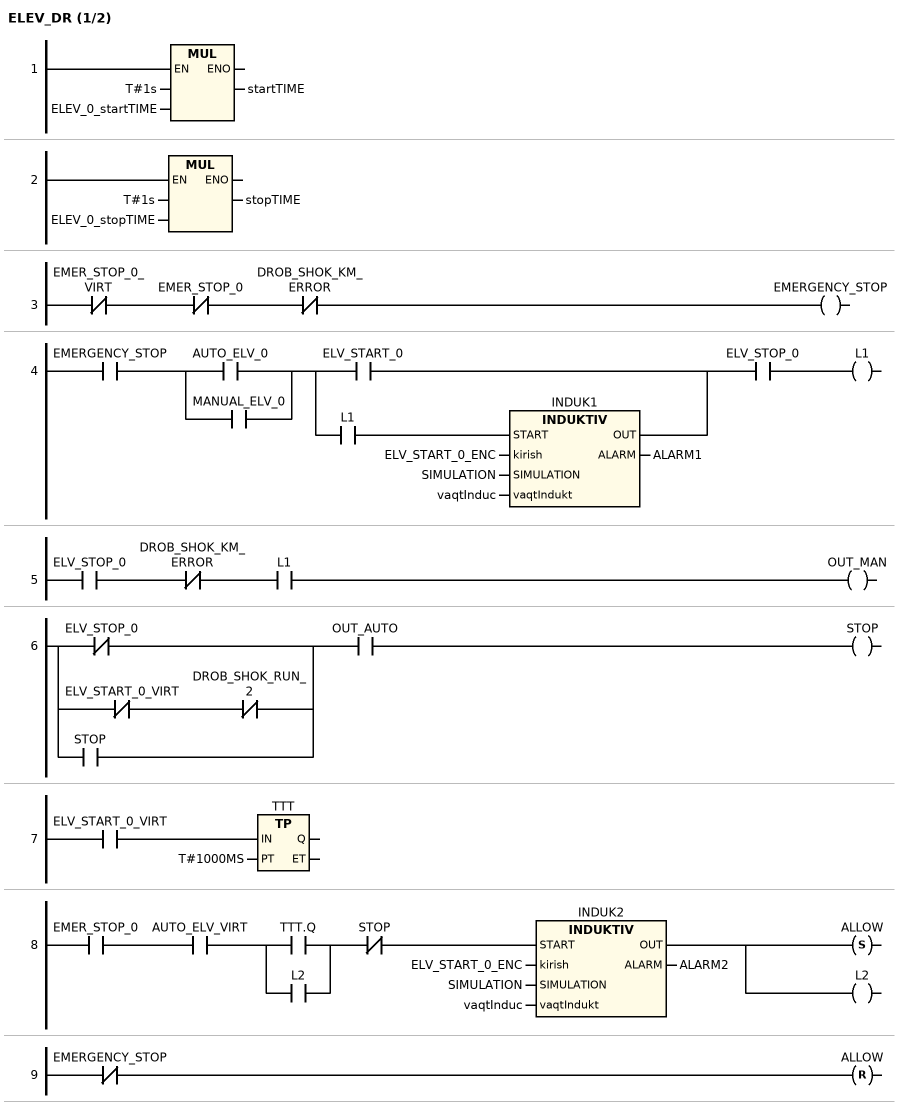
[picture p48: ELEV_DR (LD)]
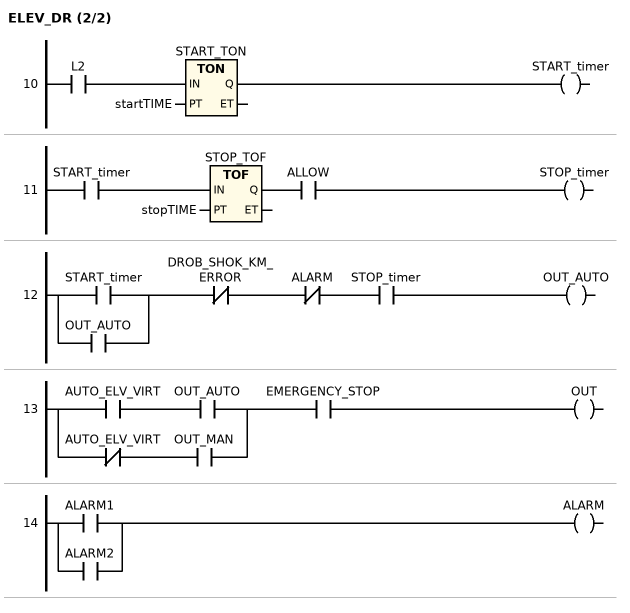
_LD_ (* Ladder Diagram *)
NETWORK 1
	*
		EN --- MUL(T#1s, ELEV_0_startTIME) => startTIME
NETWORK 2
	*
		EN --- MUL(T#1s, ELEV_0_stopTIME) => stopTIME
NETWORK 3
	[/EMER_STOP_0_VIRT] - [/EMER_STOP_0] - [/DROB_SHOK_KM_ERROR] --- (EMERGENCY_STOP)
NETWORK 4
	[EMERGENCY_STOP] - { [AUTO_ELV_0] | [MANUAL_ELV_0] } - { [ELV_START_0] | [L1] - INDUK1:INDUKTIV(START: *, kirish: ELV_START_0_ENC, SIMULATION: SIMULATION, vaqtIndukt: vaqtInduc, ALARM => ALARM1) } - [ELV_STOP_0] --- (L1)
NETWORK 5
	[ELV_STOP_0] - [/DROB_SHOK_KM_ERROR] - [L1] --- (OUT_MAN)
NETWORK 6
	{ [/ELV_STOP_0] | [/ELV_START_0_VIRT] - [/DROB_SHOK_RUN_2] | [STOP] } - [OUT_AUTO] --- (STOP)
NETWORK 7
	[ELV_START_0_VIRT] - TTT:TP(IN: *, PT: T#1000MS)
NETWORK 8
	[EMER_STOP_0] - [AUTO_ELV_VIRT] - { [TTT.Q] | [L2] } - [/STOP] - INDUK2:INDUKTIV(START: *, kirish: ELV_START_0_ENC, SIMULATION: SIMULATION, vaqtIndukt: vaqtInduc, ALARM => ALARM2) --- (S ALLOW) (L2)
NETWORK 9
	[/EMERGENCY_STOP] --- (R ALLOW)
NETWORK 10
	[L2] - START_TON:TON(IN: *, PT: startTIME) --- (START_timer)
NETWORK 11
	[START_timer] - STOP_TOF:TOF(IN: *, PT: stopTIME) - [ALLOW] --- (STOP_timer)
NETWORK 12
	{ [START_timer] | [OUT_AUTO] } - [/DROB_SHOK_KM_ERROR] - [/ALARM] - [STOP_timer] --- (OUT_AUTO)
NETWORK 13
	{ [AUTO_ELV_VIRT] - [OUT_AUTO] | [/AUTO_ELV_VIRT] - [OUT_MAN] } - [EMERGENCY_STOP] --- (OUT)
NETWORK 14
	{ [ALARM1] | [ALARM2] } --- (ALARM)
_END_LD_
(* the same logic as Structured Text *)
(* Network 1 *)
startTIME := T#1s * ELEV_0_startTIME;
(* Network 2 *)
stopTIME := T#1s * ELEV_0_stopTIME;
(* Network 3 *)
EMERGENCY_STOP := NOT EMER_STOP_0_VIRT AND NOT EMER_STOP_0 AND NOT DROB_SHOK_KM_ERROR;
(* Network 4 *)
_p1 := EMERGENCY_STOP AND (AUTO_ELV_0 OR MANUAL_ELV_0);
INDUK1(START := _p1 AND L1, kirish := ELV_START_0_ENC, SIMULATION := SIMULATION, vaqtIndukt := vaqtInduc);
ALARM1 := INDUK1.ALARM;
L1 := (_p1 AND ELV_START_0 OR INDUK1.OUT) AND ELV_STOP_0;
(* Network 5 *)
OUT_MAN := ELV_STOP_0 AND NOT DROB_SHOK_KM_ERROR AND L1;
(* Network 6 *)
STOP := (NOT ELV_STOP_0 OR NOT ELV_START_0_VIRT AND NOT DROB_SHOK_RUN_2 OR STOP) AND OUT_AUTO;
(* Network 7 *)
TTT(IN := ELV_START_0_VIRT, PT := T#1000MS);
(* Network 8 *)
INDUK2(START := EMER_STOP_0 AND AUTO_ELV_VIRT AND (TTT.Q OR L2) AND NOT STOP, kirish := ELV_START_0_ENC, SIMULATION := SIMULATION, vaqtIndukt := vaqtInduc);
ALARM2 := INDUK2.ALARM;
IF INDUK2.OUT THEN ALLOW := TRUE; END_IF;
L2 := INDUK2.OUT;
(* Network 9 *)
IF NOT EMERGENCY_STOP THEN ALLOW := FALSE; END_IF;
(* Network 10 *)
START_TON(IN := L2, PT := startTIME);
START_timer := START_TON.Q;
(* Network 11 *)
STOP_TOF(IN := START_timer, PT := stopTIME);
STOP_timer := STOP_TOF.Q AND ALLOW;
(* Network 12 *)
OUT_AUTO := (START_timer OR OUT_AUTO) AND NOT DROB_SHOK_KM_ERROR AND NOT ALARM AND STOP_timer;
(* Network 13 *)
OUT := (AUTO_ELV_VIRT AND OUT_AUTO OR NOT AUTO_ELV_VIRT AND OUT_MAN) AND EMERGENCY_STOP;
(* Network 14 *)
ALARM := ALARM1 OR ALARM2;
END_FUNCTION_BLOCK

(* POU DROBILKA2, LD *)
PROGRAM DROBILKA2
VAR
	convTON : TON;
	conVAQT : TIME := T#180s;
	drobTON : TON;
	drobVAQT: TIME := T#180s;
	maxTON : TON;
	maxVAQT: TIME := T#5s;
	ELV_F_TRIG: F_TRIG;
	TANK_FULL: BOOL;
	ELV_R_TRIG: R_TRIG;
END_VAR
VAR (* helpers for the ST form of the networks *)
	_p1 : BOOL;
END_VAR
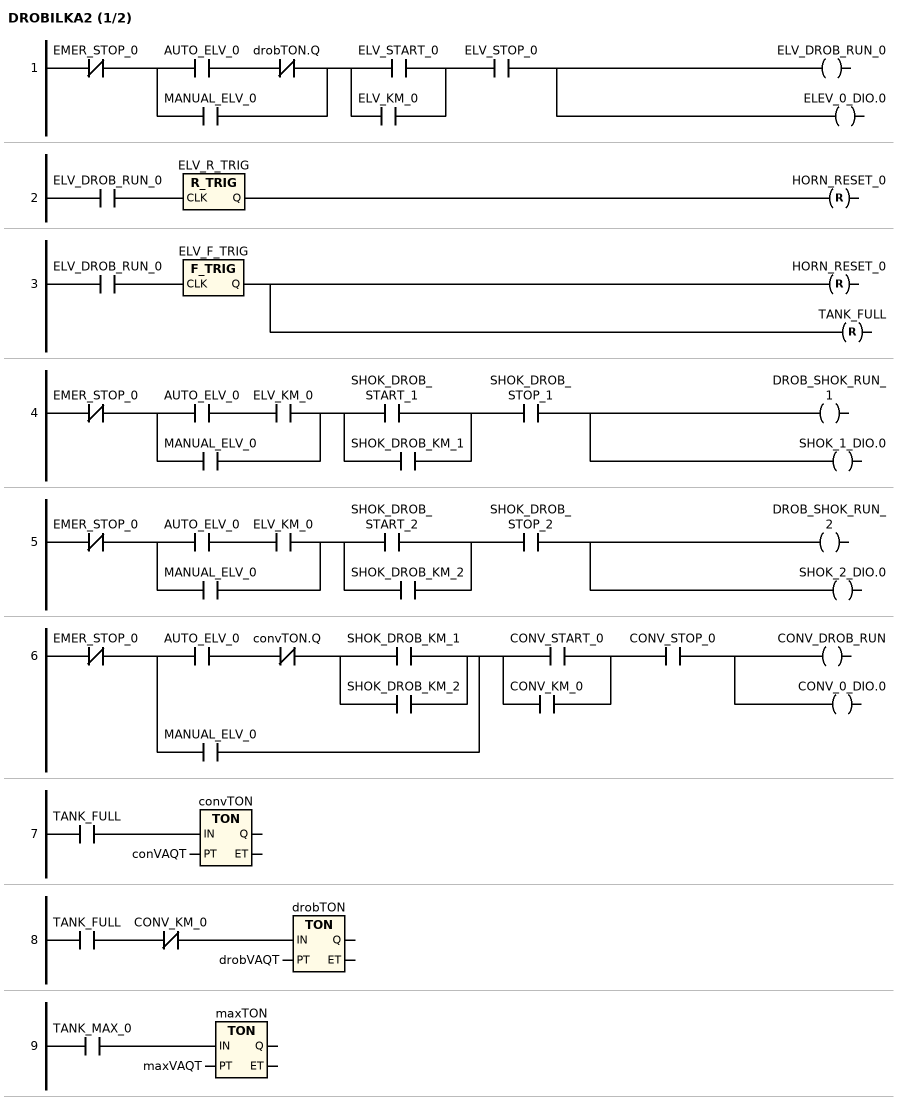
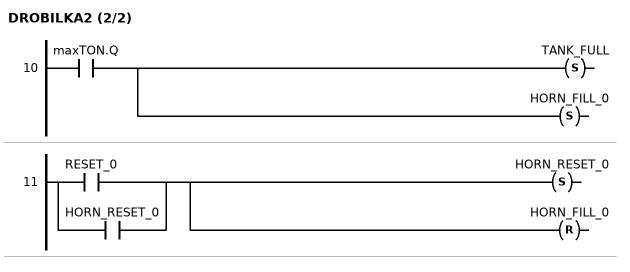
_LD_ (* Ladder Diagram *)
NETWORK 1
	[/EMER_STOP_0] - { [AUTO_ELV_0] - [/drobTON.Q] | [MANUAL_ELV_0] } - { [ELV_START_0] | [ELV_KM_0] } - [ELV_STOP_0] --- (ELV_DROB_RUN_0) (ELEV_0_DIO.0)
NETWORK 2
	[ELV_DROB_RUN_0] - ELV_R_TRIG:R_TRIG(CLK: *) --- (R HORN_RESET_0)
NETWORK 3
	[ELV_DROB_RUN_0] - ELV_F_TRIG:F_TRIG(CLK: *) --- (R HORN_RESET_0) (R TANK_FULL)
NETWORK 4
	[/EMER_STOP_0] - { [AUTO_ELV_0] - [ELV_KM_0] | [MANUAL_ELV_0] } - { [SHOK_DROB_START_1] | [SHOK_DROB_KM_1] } - [SHOK_DROB_STOP_1] --- (DROB_SHOK_RUN_1) (SHOK_1_DIO.0)
NETWORK 5
	[/EMER_STOP_0] - { [AUTO_ELV_0] - [ELV_KM_0] | [MANUAL_ELV_0] } - { [SHOK_DROB_START_2] | [SHOK_DROB_KM_2] } - [SHOK_DROB_STOP_2] --- (DROB_SHOK_RUN_2) (SHOK_2_DIO.0)
NETWORK 6
	[/EMER_STOP_0] - { [AUTO_ELV_0] - [/convTON.Q] - { [SHOK_DROB_KM_1] | [SHOK_DROB_KM_2] } | [MANUAL_ELV_0] } - { [CONV_START_0] | [CONV_KM_0] } - [CONV_STOP_0] --- (CONV_DROB_RUN) (CONV_0_DIO.0)
NETWORK 7
	[TANK_FULL] - convTON:TON(IN: *, PT: conVAQT)
NETWORK 8
	[TANK_FULL] - [/CONV_KM_0] - drobTON:TON(IN: *, PT: drobVAQT)
NETWORK 9
	[TANK_MAX_0] - maxTON:TON(IN: *, PT: maxVAQT)
NETWORK 10
	[maxTON.Q] --- (S TANK_FULL) (S HORN_FILL_0)
NETWORK 11
	{ [RESET_0] | [HORN_RESET_0] } --- (S HORN_RESET_0) (R HORN_FILL_0)
_END_LD_
(* the same logic as Structured Text *)
(* Network 1 *)
ELV_DROB_RUN_0 := NOT EMER_STOP_0 AND (AUTO_ELV_0 AND NOT drobTON.Q OR MANUAL_ELV_0) AND (ELV_START_0 OR ELV_KM_0) AND ELV_STOP_0;
ELEV_0_DIO.0 := ELV_DROB_RUN_0;
(* Network 2 *)
ELV_R_TRIG(CLK := ELV_DROB_RUN_0);
IF ELV_R_TRIG.Q THEN HORN_RESET_0 := FALSE; END_IF;
(* Network 3 *)
ELV_F_TRIG(CLK := ELV_DROB_RUN_0);
IF ELV_F_TRIG.Q THEN HORN_RESET_0 := FALSE; TANK_FULL := FALSE; END_IF;
(* Network 4 *)
DROB_SHOK_RUN_1 := NOT EMER_STOP_0 AND (AUTO_ELV_0 AND ELV_KM_0 OR MANUAL_ELV_0) AND (SHOK_DROB_START_1 OR SHOK_DROB_KM_1) AND SHOK_DROB_STOP_1;
SHOK_1_DIO.0 := DROB_SHOK_RUN_1;
(* Network 5 *)
DROB_SHOK_RUN_2 := NOT EMER_STOP_0 AND (AUTO_ELV_0 AND ELV_KM_0 OR MANUAL_ELV_0) AND (SHOK_DROB_START_2 OR SHOK_DROB_KM_2) AND SHOK_DROB_STOP_2;
SHOK_2_DIO.0 := DROB_SHOK_RUN_2;
(* Network 6 *)
CONV_DROB_RUN := NOT EMER_STOP_0 AND (AUTO_ELV_0 AND NOT convTON.Q AND (SHOK_DROB_KM_1 OR SHOK_DROB_KM_2) OR MANUAL_ELV_0) AND (CONV_START_0 OR CONV_KM_0) AND CONV_STOP_0;
CONV_0_DIO.0 := CONV_DROB_RUN;
(* Network 7 *)
convTON(IN := TANK_FULL, PT := conVAQT);
(* Network 8 *)
drobTON(IN := TANK_FULL AND NOT CONV_KM_0, PT := drobVAQT);
(* Network 9 *)
maxTON(IN := TANK_MAX_0, PT := maxVAQT);
(* Network 10 *)
IF maxTON.Q THEN TANK_FULL := TRUE; HORN_FILL_0 := TRUE; END_IF;
(* Network 11 *)
_p1 := RESET_0 OR HORN_RESET_0;
IF _p1 THEN HORN_RESET_0 := TRUE; HORN_FILL_0 := FALSE; END_IF;
END_PROGRAM

(* POU main_1212, LD *)
PROGRAM main_1212
VAR
	MAH_YET3 : BOOL;
	VAQT : TIME := T#10s;
       VAQT1: TIME := T#4s;
       VAQT2 : TIME := T#6s;
      VAQT3 : TIME := T#6s;
	vaqtInduc : WORD := 15;
	VIBRATOR3_T: BOOL;
	TON1: TON;
	TON2: TON;
	OUT: BOOL;
	IND1: INDUKTIV;
	IND2: INDUKTIV;


	STOP: BOOL;
	CHIQSH: BOOL;
	PUSK: BOOL;
	MAH_YET4: BOOL;
	VIBRATOR4_T: BOOL;
	induk: BOOL;

	ALR_ELEV1: BOOL;
	ALR_ELEV2: BOOL;
	ALR_ELEV3: BOOL;
	ALR_ELEV4: BOOL;
	IND_ELV_1: INDUKTIV;
	IND_SHNK_3: INDUKTIV;
	IND_SHNK_4: INDUKTIV;
	IND_SHNK_SKL_4: INDUKTIV;
	IND_SEPR_4: INDUKTIV;
	IND_MILL_3: INDUKTIV;
	IND_MILL_4: INDUKTIV;

END_VAR
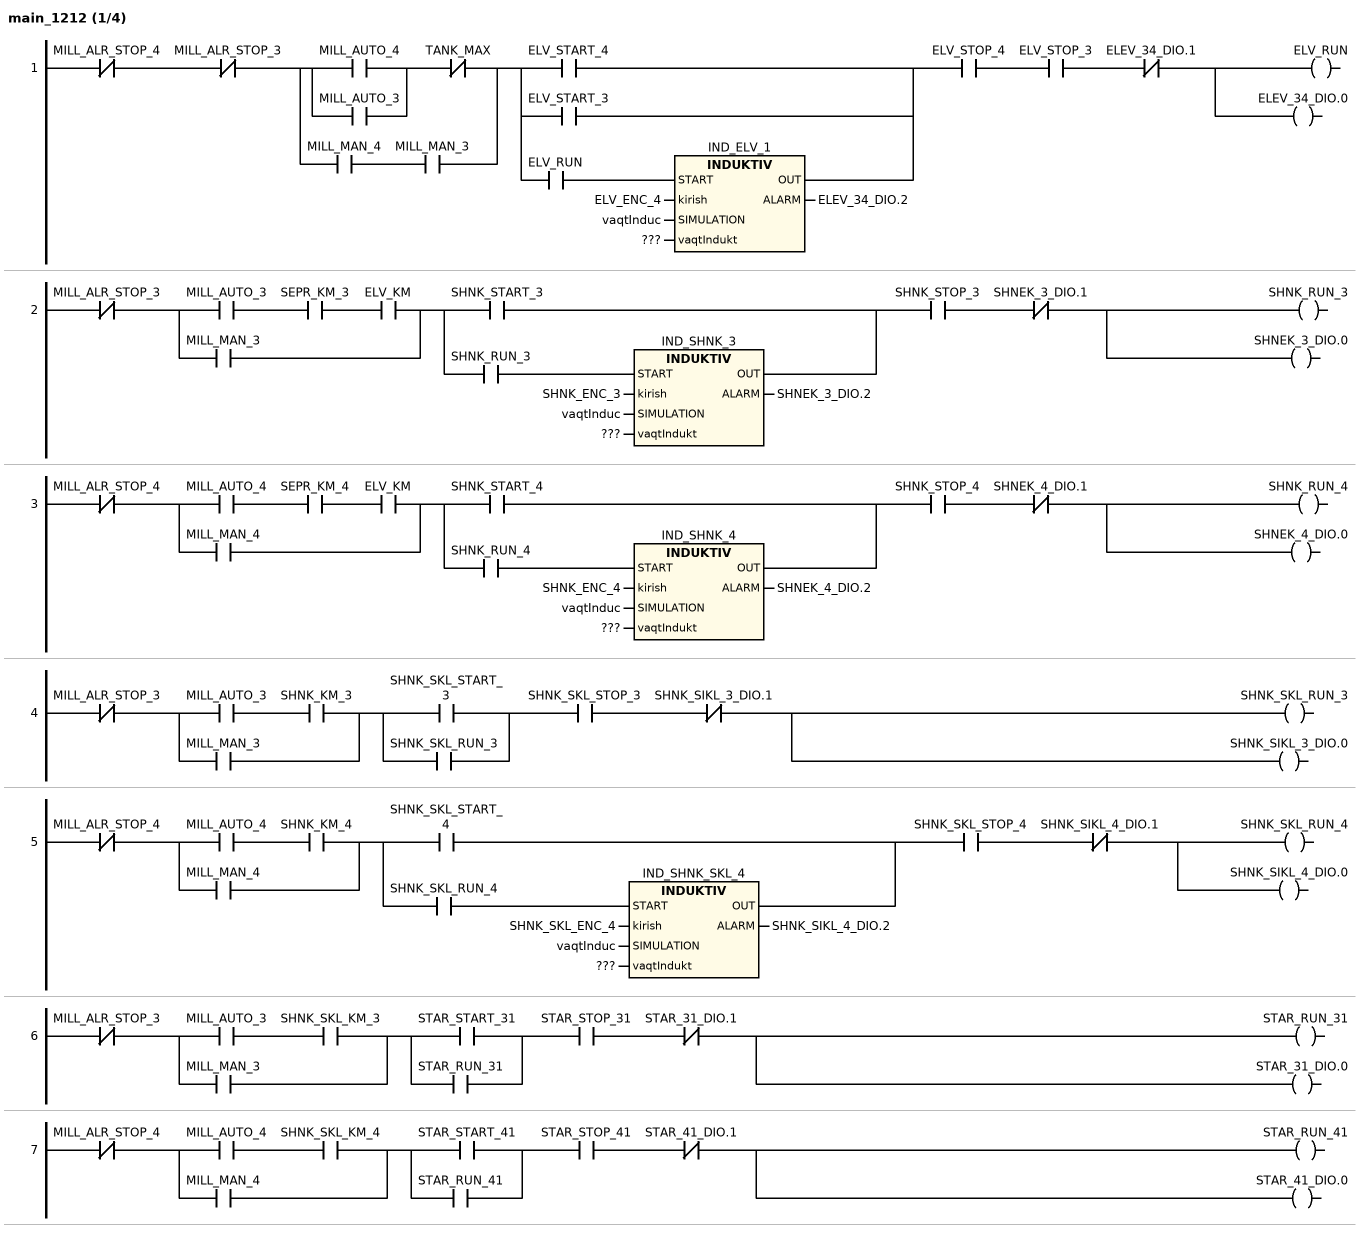
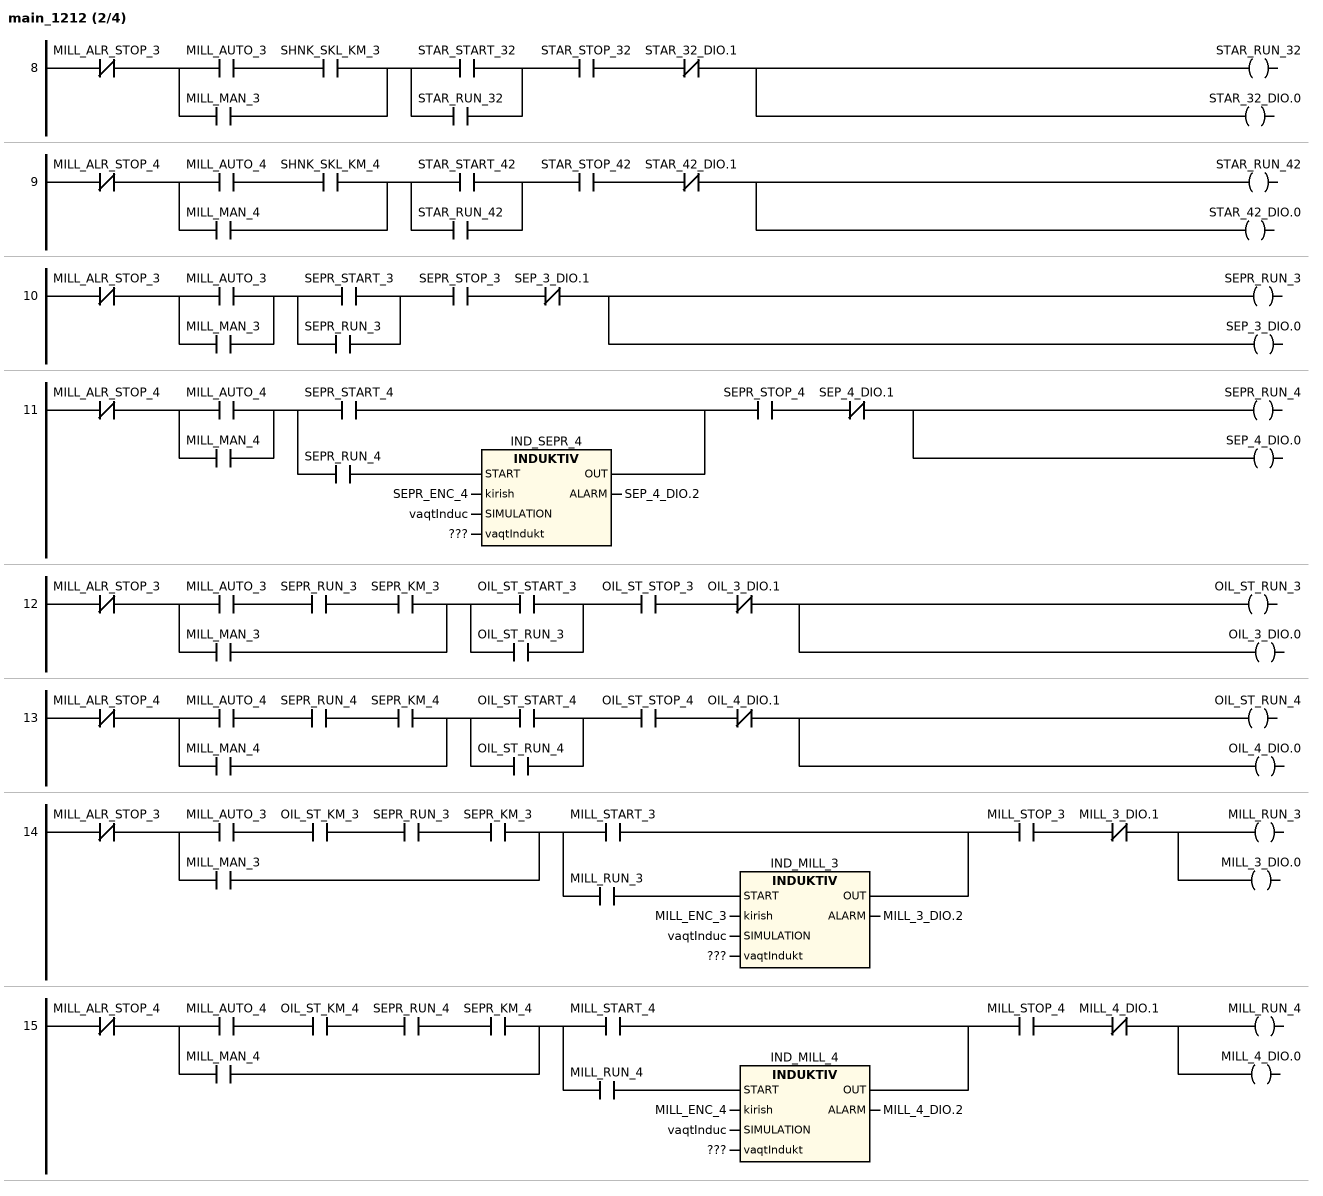
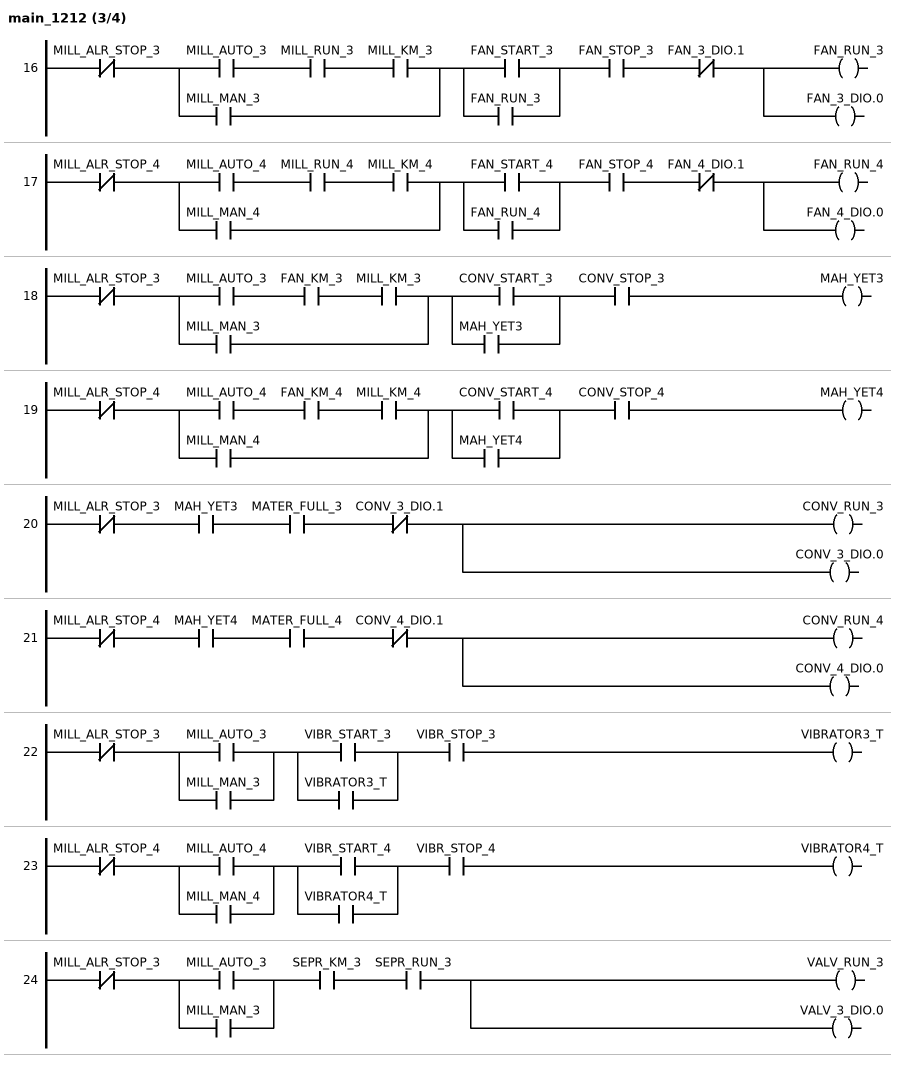
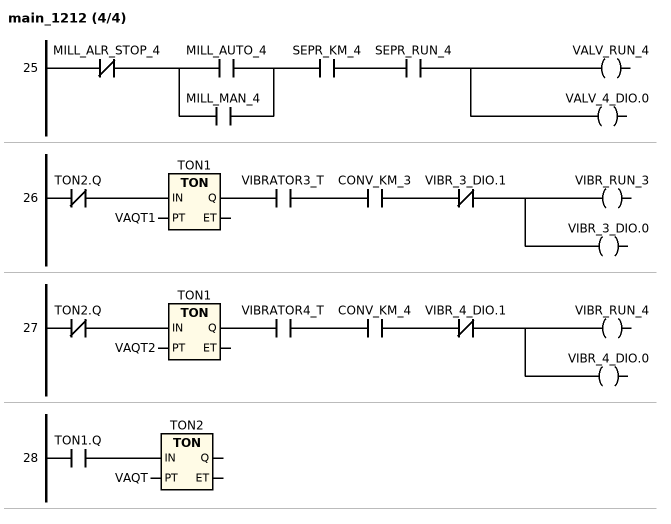
_LD_ (* Ladder Diagram *)
NETWORK 1
	[/MILL_ALR_STOP_4] - [/MILL_ALR_STOP_3] - { { [MILL_AUTO_4] | [MILL_AUTO_3] } - [/TANK_MAX] | [MILL_MAN_4] - [MILL_MAN_3] } - { [ELV_START_4] | [ELV_START_3] | [ELV_RUN] - IND_ELV_1:INDUKTIV(START: *, kirish: ELV_ENC_4, SIMULATION: vaqtInduc, vaqtIndukt: ???, ALARM => ELEV_34_DIO.2) } - [ELV_STOP_4] - [ELV_STOP_3] - [/ELEV_34_DIO.1] --- (ELV_RUN) (ELEV_34_DIO.0)
NETWORK 2
	[/MILL_ALR_STOP_3] - { [MILL_AUTO_3] - [SEPR_KM_3] - [ELV_KM] | [MILL_MAN_3] } - { [SHNK_START_3] | [SHNK_RUN_3] - IND_SHNK_3:INDUKTIV(START: *, kirish: SHNK_ENC_3, SIMULATION: vaqtInduc, vaqtIndukt: ???, ALARM => SHNEK_3_DIO.2) } - [SHNK_STOP_3] - [/SHNEK_3_DIO.1] --- (SHNK_RUN_3) (SHNEK_3_DIO.0)
NETWORK 3
	[/MILL_ALR_STOP_4] - { [MILL_AUTO_4] - [SEPR_KM_4] - [ELV_KM] | [MILL_MAN_4] } - { [SHNK_START_4] | [SHNK_RUN_4] - IND_SHNK_4:INDUKTIV(START: *, kirish: SHNK_ENC_4, SIMULATION: vaqtInduc, vaqtIndukt: ???, ALARM => SHNEK_4_DIO.2) } - [SHNK_STOP_4] - [/SHNEK_4_DIO.1] --- (SHNK_RUN_4) (SHNEK_4_DIO.0)
NETWORK 4
	[/MILL_ALR_STOP_3] - { [MILL_AUTO_3] - [SHNK_KM_3] | [MILL_MAN_3] } - { [SHNK_SKL_START_3] | [SHNK_SKL_RUN_3] } - [SHNK_SKL_STOP_3] - [/SHNK_SIKL_3_DIO.1] --- (SHNK_SKL_RUN_3) (SHNK_SIKL_3_DIO.0)
NETWORK 5
	[/MILL_ALR_STOP_4] - { [MILL_AUTO_4] - [SHNK_KM_4] | [MILL_MAN_4] } - { [SHNK_SKL_START_4] | [SHNK_SKL_RUN_4] - IND_SHNK_SKL_4:INDUKTIV(START: *, kirish: SHNK_SKL_ENC_4, SIMULATION: vaqtInduc, vaqtIndukt: ???, ALARM => SHNK_SIKL_4_DIO.2) } - [SHNK_SKL_STOP_4] - [/SHNK_SIKL_4_DIO.1] --- (SHNK_SKL_RUN_4) (SHNK_SIKL_4_DIO.0)
NETWORK 6
	[/MILL_ALR_STOP_3] - { [MILL_AUTO_3] - [SHNK_SKL_KM_3] | [MILL_MAN_3] } - { [STAR_START_31] | [STAR_RUN_31] } - [STAR_STOP_31] - [/STAR_31_DIO.1] --- (STAR_RUN_31) (STAR_31_DIO.0)
NETWORK 7
	[/MILL_ALR_STOP_4] - { [MILL_AUTO_4] - [SHNK_SKL_KM_4] | [MILL_MAN_4] } - { [STAR_START_41] | [STAR_RUN_41] } - [STAR_STOP_41] - [/STAR_41_DIO.1] --- (STAR_RUN_41) (STAR_41_DIO.0)
NETWORK 8
	[/MILL_ALR_STOP_3] - { [MILL_AUTO_3] - [SHNK_SKL_KM_3] | [MILL_MAN_3] } - { [STAR_START_32] | [STAR_RUN_32] } - [STAR_STOP_32] - [/STAR_32_DIO.1] --- (STAR_RUN_32) (STAR_32_DIO.0)
NETWORK 9
	[/MILL_ALR_STOP_4] - { [MILL_AUTO_4] - [SHNK_SKL_KM_4] | [MILL_MAN_4] } - { [STAR_START_42] | [STAR_RUN_42] } - [STAR_STOP_42] - [/STAR_42_DIO.1] --- (STAR_RUN_42) (STAR_42_DIO.0)
NETWORK 10
	[/MILL_ALR_STOP_3] - { [MILL_AUTO_3] | [MILL_MAN_3] } - { [SEPR_START_3] | [SEPR_RUN_3] } - [SEPR_STOP_3] - [/SEP_3_DIO.1] --- (SEPR_RUN_3) (SEP_3_DIO.0)
NETWORK 11
	[/MILL_ALR_STOP_4] - { [MILL_AUTO_4] | [MILL_MAN_4] } - { [SEPR_START_4] | [SEPR_RUN_4] - IND_SEPR_4:INDUKTIV(START: *, kirish: SEPR_ENC_4, SIMULATION: vaqtInduc, vaqtIndukt: ???, ALARM => SEP_4_DIO.2) } - [SEPR_STOP_4] - [/SEP_4_DIO.1] --- (SEPR_RUN_4) (SEP_4_DIO.0)
NETWORK 12
	[/MILL_ALR_STOP_3] - { [MILL_AUTO_3] - [SEPR_RUN_3] - [SEPR_KM_3] | [MILL_MAN_3] } - { [OIL_ST_START_3] | [OIL_ST_RUN_3] } - [OIL_ST_STOP_3] - [/OIL_3_DIO.1] --- (OIL_ST_RUN_3) (OIL_3_DIO.0)
NETWORK 13
	[/MILL_ALR_STOP_4] - { [MILL_AUTO_4] - [SEPR_RUN_4] - [SEPR_KM_4] | [MILL_MAN_4] } - { [OIL_ST_START_4] | [OIL_ST_RUN_4] } - [OIL_ST_STOP_4] - [/OIL_4_DIO.1] --- (OIL_ST_RUN_4) (OIL_4_DIO.0)
NETWORK 14
	[/MILL_ALR_STOP_3] - { [MILL_AUTO_3] - [OIL_ST_KM_3] - [SEPR_RUN_3] - [SEPR_KM_3] | [MILL_MAN_3] } - { [MILL_START_3] | [MILL_RUN_3] - IND_MILL_3:INDUKTIV(START: *, kirish: MILL_ENC_3, SIMULATION: vaqtInduc, vaqtIndukt: ???, ALARM => MILL_3_DIO.2) } - [MILL_STOP_3] - [/MILL_3_DIO.1] --- (MILL_RUN_3) (MILL_3_DIO.0)
NETWORK 15
	[/MILL_ALR_STOP_4] - { [MILL_AUTO_4] - [OIL_ST_KM_4] - [SEPR_RUN_4] - [SEPR_KM_4] | [MILL_MAN_4] } - { [MILL_START_4] | [MILL_RUN_4] - IND_MILL_4:INDUKTIV(START: *, kirish: MILL_ENC_4, SIMULATION: vaqtInduc, vaqtIndukt: ???, ALARM => MILL_4_DIO.2) } - [MILL_STOP_4] - [/MILL_4_DIO.1] --- (MILL_RUN_4) (MILL_4_DIO.0)
NETWORK 16
	[/MILL_ALR_STOP_3] - { [MILL_AUTO_3] - [MILL_RUN_3] - [MILL_KM_3] | [MILL_MAN_3] } - { [FAN_START_3] | [FAN_RUN_3] } - [FAN_STOP_3] - [/FAN_3_DIO.1] --- (FAN_RUN_3) (FAN_3_DIO.0)
NETWORK 17
	[/MILL_ALR_STOP_4] - { [MILL_AUTO_4] - [MILL_RUN_4] - [MILL_KM_4] | [MILL_MAN_4] } - { [FAN_START_4] | [FAN_RUN_4] } - [FAN_STOP_4] - [/FAN_4_DIO.1] --- (FAN_RUN_4) (FAN_4_DIO.0)
NETWORK 18
	[/MILL_ALR_STOP_3] - { [MILL_AUTO_3] - [FAN_KM_3] - [MILL_KM_3] | [MILL_MAN_3] } - { [CONV_START_3] | [MAH_YET3] } - [CONV_STOP_3] --- (MAH_YET3)
NETWORK 19
	[/MILL_ALR_STOP_4] - { [MILL_AUTO_4] - [FAN_KM_4] - [MILL_KM_4] | [MILL_MAN_4] } - { [CONV_START_4] | [MAH_YET4] } - [CONV_STOP_4] --- (MAH_YET4)
NETWORK 20
	[/MILL_ALR_STOP_3] - [MAH_YET3] - [MATER_FULL_3] - [/CONV_3_DIO.1] --- (CONV_RUN_3) (CONV_3_DIO.0)
NETWORK 21
	[/MILL_ALR_STOP_4] - [MAH_YET4] - [MATER_FULL_4] - [/CONV_4_DIO.1] --- (CONV_RUN_4) (CONV_4_DIO.0)
NETWORK 22
	[/MILL_ALR_STOP_3] - { [MILL_AUTO_3] | [MILL_MAN_3] } - { [VIBR_START_3] | [VIBRATOR3_T] } - [VIBR_STOP_3] --- (VIBRATOR3_T)
NETWORK 23
	[/MILL_ALR_STOP_4] - { [MILL_AUTO_4] | [MILL_MAN_4] } - { [VIBR_START_4] | [VIBRATOR4_T] } - [VIBR_STOP_4] --- (VIBRATOR4_T)
NETWORK 24
	[/MILL_ALR_STOP_3] - { [MILL_AUTO_3] | [MILL_MAN_3] } - [SEPR_KM_3] - [SEPR_RUN_3] --- (VALV_RUN_3) (VALV_3_DIO.0)
NETWORK 25
	[/MILL_ALR_STOP_4] - { [MILL_AUTO_4] | [MILL_MAN_4] } - [SEPR_KM_4] - [SEPR_RUN_4] --- (VALV_RUN_4) (VALV_4_DIO.0)
NETWORK 26
	[/TON2.Q] - TON1:TON(IN: *, PT: VAQT1) - [VIBRATOR3_T] - [CONV_KM_3] - [/VIBR_3_DIO.1] --- (VIBR_RUN_3) (VIBR_3_DIO.0)
NETWORK 27
	[/TON2.Q] - TON1:TON(IN: *, PT: VAQT2) - [VIBRATOR4_T] - [CONV_KM_4] - [/VIBR_4_DIO.1] --- (VIBR_RUN_4) (VIBR_4_DIO.0)
NETWORK 28
	[TON1.Q] - TON2:TON(IN: *, PT: VAQT)
_END_LD_
(* the same logic as Structured Text *)
(* Network 1: see the listing above *)
(* Network 2: see the listing above *)
(* Network 3: see the listing above *)
(* Network 4 *)
SHNK_SKL_RUN_3 := NOT MILL_ALR_STOP_3 AND (MILL_AUTO_3 AND SHNK_KM_3 OR MILL_MAN_3) AND (SHNK_SKL_START_3 OR SHNK_SKL_RUN_3) AND SHNK_SKL_STOP_3 AND NOT SHNK_SIKL_3_DIO.1;
SHNK_SIKL_3_DIO.0 := SHNK_SKL_RUN_3;
(* Network 5: see the listing above *)
(* Network 6 *)
STAR_RUN_31 := NOT MILL_ALR_STOP_3 AND (MILL_AUTO_3 AND SHNK_SKL_KM_3 OR MILL_MAN_3) AND (STAR_START_31 OR STAR_RUN_31) AND STAR_STOP_31 AND NOT STAR_31_DIO.1;
STAR_31_DIO.0 := STAR_RUN_31;
(* Network 7 *)
STAR_RUN_41 := NOT MILL_ALR_STOP_4 AND (MILL_AUTO_4 AND SHNK_SKL_KM_4 OR MILL_MAN_4) AND (STAR_START_41 OR STAR_RUN_41) AND STAR_STOP_41 AND NOT STAR_41_DIO.1;
STAR_41_DIO.0 := STAR_RUN_41;
(* Network 8 *)
STAR_RUN_32 := NOT MILL_ALR_STOP_3 AND (MILL_AUTO_3 AND SHNK_SKL_KM_3 OR MILL_MAN_3) AND (STAR_START_32 OR STAR_RUN_32) AND STAR_STOP_32 AND NOT STAR_32_DIO.1;
STAR_32_DIO.0 := STAR_RUN_32;
(* Network 9 *)
STAR_RUN_42 := NOT MILL_ALR_STOP_4 AND (MILL_AUTO_4 AND SHNK_SKL_KM_4 OR MILL_MAN_4) AND (STAR_START_42 OR STAR_RUN_42) AND STAR_STOP_42 AND NOT STAR_42_DIO.1;
STAR_42_DIO.0 := STAR_RUN_42;
(* Network 10 *)
SEPR_RUN_3 := NOT MILL_ALR_STOP_3 AND (MILL_AUTO_3 OR MILL_MAN_3) AND (SEPR_START_3 OR SEPR_RUN_3) AND SEPR_STOP_3 AND NOT SEP_3_DIO.1;
SEP_3_DIO.0 := SEPR_RUN_3;
(* Network 11: see the listing above *)
(* Network 12 *)
OIL_ST_RUN_3 := NOT MILL_ALR_STOP_3 AND (MILL_AUTO_3 AND SEPR_RUN_3 AND SEPR_KM_3 OR MILL_MAN_3) AND (OIL_ST_START_3 OR OIL_ST_RUN_3) AND OIL_ST_STOP_3 AND NOT OIL_3_DIO.1;
OIL_3_DIO.0 := OIL_ST_RUN_3;
(* Network 13 *)
OIL_ST_RUN_4 := NOT MILL_ALR_STOP_4 AND (MILL_AUTO_4 AND SEPR_RUN_4 AND SEPR_KM_4 OR MILL_MAN_4) AND (OIL_ST_START_4 OR OIL_ST_RUN_4) AND OIL_ST_STOP_4 AND NOT OIL_4_DIO.1;
OIL_4_DIO.0 := OIL_ST_RUN_4;
(* Network 14: see the listing above *)
(* Network 15: see the listing above *)
(* Network 16 *)
FAN_RUN_3 := NOT MILL_ALR_STOP_3 AND (MILL_AUTO_3 AND MILL_RUN_3 AND MILL_KM_3 OR MILL_MAN_3) AND (FAN_START_3 OR FAN_RUN_3) AND FAN_STOP_3 AND NOT FAN_3_DIO.1;
FAN_3_DIO.0 := FAN_RUN_3;
(* Network 17 *)
FAN_RUN_4 := NOT MILL_ALR_STOP_4 AND (MILL_AUTO_4 AND MILL_RUN_4 AND MILL_KM_4 OR MILL_MAN_4) AND (FAN_START_4 OR FAN_RUN_4) AND FAN_STOP_4 AND NOT FAN_4_DIO.1;
FAN_4_DIO.0 := FAN_RUN_4;
(* Network 18 *)
MAH_YET3 := NOT MILL_ALR_STOP_3 AND (MILL_AUTO_3 AND FAN_KM_3 AND MILL_KM_3 OR MILL_MAN_3) AND (CONV_START_3 OR MAH_YET3) AND CONV_STOP_3;
(* Network 19 *)
MAH_YET4 := NOT MILL_ALR_STOP_4 AND (MILL_AUTO_4 AND FAN_KM_4 AND MILL_KM_4 OR MILL_MAN_4) AND (CONV_START_4 OR MAH_YET4) AND CONV_STOP_4;
(* Network 20 *)
CONV_RUN_3 := NOT MILL_ALR_STOP_3 AND MAH_YET3 AND MATER_FULL_3 AND NOT CONV_3_DIO.1;
CONV_3_DIO.0 := CONV_RUN_3;
(* Network 21 *)
CONV_RUN_4 := NOT MILL_ALR_STOP_4 AND MAH_YET4 AND MATER_FULL_4 AND NOT CONV_4_DIO.1;
CONV_4_DIO.0 := CONV_RUN_4;
(* Network 22 *)
VIBRATOR3_T := NOT MILL_ALR_STOP_3 AND (MILL_AUTO_3 OR MILL_MAN_3) AND (VIBR_START_3 OR VIBRATOR3_T) AND VIBR_STOP_3;
(* Network 23 *)
VIBRATOR4_T := NOT MILL_ALR_STOP_4 AND (MILL_AUTO_4 OR MILL_MAN_4) AND (VIBR_START_4 OR VIBRATOR4_T) AND VIBR_STOP_4;
(* Network 24 *)
VALV_RUN_3 := NOT MILL_ALR_STOP_3 AND (MILL_AUTO_3 OR MILL_MAN_3) AND SEPR_KM_3 AND SEPR_RUN_3;
VALV_3_DIO.0 := VALV_RUN_3;
(* Network 25 *)
VALV_RUN_4 := NOT MILL_ALR_STOP_4 AND (MILL_AUTO_4 OR MILL_MAN_4) AND SEPR_KM_4 AND SEPR_RUN_4;
VALV_4_DIO.0 := VALV_RUN_4;
(* Network 26 *)
TON1(IN := NOT TON2.Q, PT := VAQT1);
VIBR_RUN_3 := TON1.Q AND VIBRATOR3_T AND CONV_KM_3 AND NOT VIBR_3_DIO.1;
VIBR_3_DIO.0 := VIBR_RUN_3;
(* Network 27 *)
TON1(IN := NOT TON2.Q, PT := VAQT2);
VIBR_RUN_4 := TON1.Q AND VIBRATOR4_T AND CONV_KM_4 AND NOT VIBR_4_DIO.1;
VIBR_4_DIO.0 := VIBR_RUN_4;
(* Network 28 *)
TON2(IN := TON1.Q, PT := VAQT);
END_PROGRAM

(* POU INDUKTIV_2, CFC *)
FUNCTION_BLOCK INDUKTIV_2
VAR_IN_OUT

	(*RESET : BOOL;*)

END_VAR
VAR_INPUT
	START : BOOL;
	kirish : BOOL;
	vaqtIndukt : WORD := 15;
END_VAR

VAR_OUTPUT

	OUT : BOOL;
	ALARM : BOOL;
END_VAR
VAR
	ton1: TON;
	vaqt : TIME;
	ton2: TON;
	TP1: TP;
	TP2: TP;


END_VAR
VAR (* helpers for the ST form of the networks *)
	_t11 : BOOL;
	_t41 : BOOL;
	_t47 : BOOL;
	_t44 : BOOL;
	_t45 : BOOL;
	_en19 : BOOL;
END_VAR
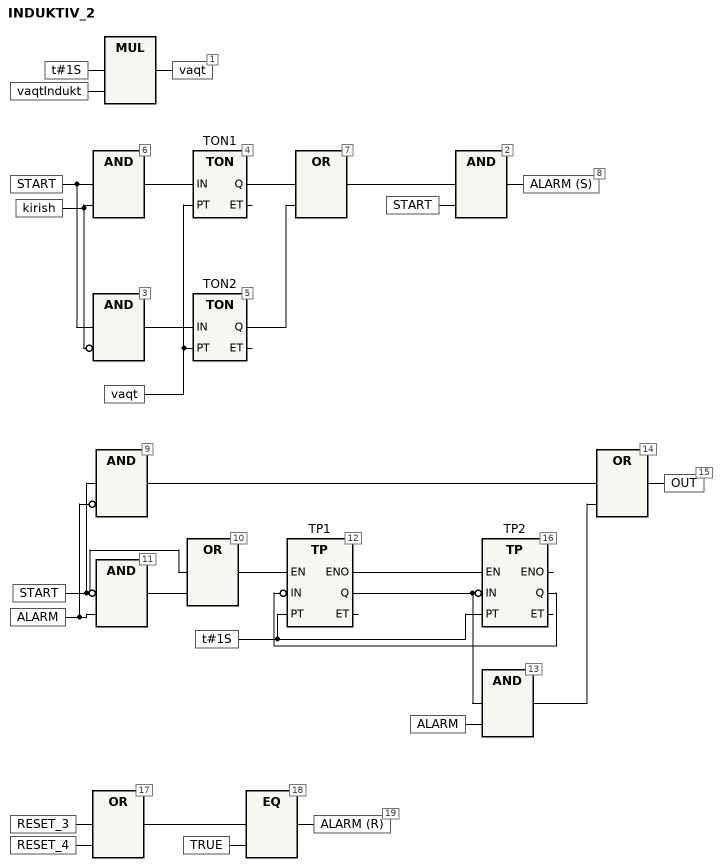
_CFC_ (* Continuous Function Chart, elements in execution order *)
#0 MUL(t#1S, vaqtIndukt)
#1 vaqt <= #0
#2 AND(#7, START)
#3 AND(START, NOT kirish)
#4 TON1:TON(IN: #6, PT: vaqt)
#5 TON2:TON(IN: #3, PT: vaqt)
#6 AND(START, kirish)
#7 OR(#4.Q, #5.Q)
#8 S ALARM <= #2
#9 AND(START, NOT ALARM)
#10 OR(START, #11)
#11 AND(NOT START, ALARM)
#12 TP1:TP(EN: #10, IN: NOT #16.Q, PT: t#1S)
#13 AND(#12.Q, ALARM)
#14 OR(#9, #13)
#15 OUT <= #14
#16 TP2:TP(EN: #12.ENO, IN: NOT #12.Q, PT: t#1S)
#17 OR(RESET_3, RESET_4)
#18 EQ(#17, TRUE)
#19 R ALARM <= #18
_END_CFC_
(* the same logic as Structured Text *)
vaqt := t#1S * vaqtIndukt;
_t41 := _t11 AND START;
TON1(IN := _t47, PT := vaqt);
TON2(IN := START AND NOT kirish, PT := vaqt);
_t47 := START AND kirish;
_t11 := TON1.Q OR TON2.Q;
IF _t41 THEN ALARM := TRUE; END_IF;
_t45 := START OR _t44;
_t44 := NOT START AND ALARM;
_en19 := _t45;
IF _en19 THEN TP1(IN := NOT TP2.Q, PT := t#1S); END_IF;
OUT := (START AND NOT ALARM) OR (TP1.Q AND ALARM);
IF _en19 THEN TP2(IN := NOT TP1.Q, PT := t#1S); END_IF;
IF (RESET_3 OR RESET_4) = TRUE THEN ALARM := FALSE; END_IF;
END_FUNCTION_BLOCK

(* POU INDUKTIV_545456, CFC *)
FUNCTION_BLOCK INDUKTIV_545456
VAR_IN_OUT

	(*RESET : BOOL;*)

END_VAR
VAR_INPUT
	START : BOOL;
	kirish : BOOL;
	vaqtIndukt : WORD := 15;
END_VAR

VAR_OUTPUT

	OUT : BOOL;
	ALARM : BOOL;
END_VAR
VAR
	ton1: TON;
	vaqt : TIME;
	ton2: TON;
	TP1: TP;
	TP2: TP;


END_VAR
VAR (* helpers for the ST form of the networks *)
	_t11 : BOOL;
	_t41 : BOOL;
	_t47 : BOOL;
END_VAR
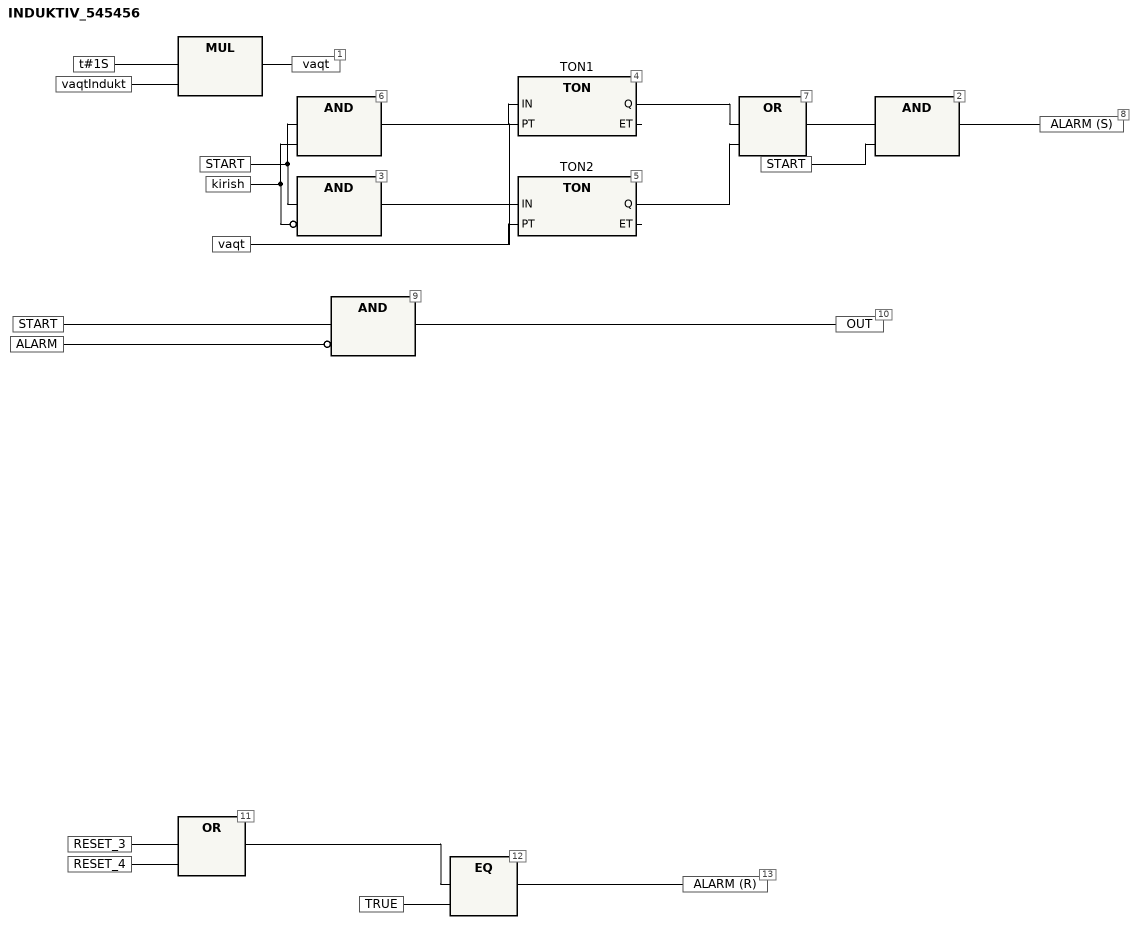
_CFC_ (* Continuous Function Chart, elements in execution order *)
#0 MUL(t#1S, vaqtIndukt)
#1 vaqt <= #0
#2 AND(#7, START)
#3 AND(START, NOT kirish)
#4 TON1:TON(IN: #6, PT: vaqt)
#5 TON2:TON(IN: #3, PT: vaqt)
#6 AND(START, kirish)
#7 OR(#4.Q, #5.Q)
#8 S ALARM <= #2
#9 AND(START, NOT ALARM)
#10 OUT <= #9
#11 OR(RESET_3, RESET_4)
#12 EQ(#11, TRUE)
#13 R ALARM <= #12
_END_CFC_
(* the same logic as Structured Text *)
vaqt := t#1S * vaqtIndukt;
_t41 := _t11 AND START;
TON1(IN := _t47, PT := vaqt);
TON2(IN := START AND NOT kirish, PT := vaqt);
_t47 := START AND kirish;
_t11 := TON1.Q OR TON2.Q;
IF _t41 THEN ALARM := TRUE; END_IF;
OUT := START AND NOT ALARM;
IF (RESET_3 OR RESET_4) = TRUE THEN ALARM := FALSE; END_IF;
END_FUNCTION_BLOCK
